{attribute 'qualified_only'}
{attribute 'strict'}
TYPE E_RunningStates :
(
	Off,
	Auto,
	Manual
);
END_TYPE

(* stored: Version 1.1.0.1, ProductVersion 3.1.4024.12
   DUT E_RunningStates: Id {9b8256c7-17b8-4c37-adab-17e648d60200} *)
